// TIA Portal project "机器人" (V14)

(* hardware
DEVICE "S71500/ET200MP station_1"  S7-1500 station
   slot 0: "导轨_0"  Rack  6ES7 590-1***0-0AA0
   slot 1: "PLC_1"  CPU 1516-3 PN/DP  6ES7 516-3AN01-0AB0  V2.1
      slot 3: "CPU 显示_1"  6ES7591-1BA00-0AA0
   slot 2: "DI 32x24VDC HF_1"  DI 32x24VDC HF  6ES7 521-1BL00-0AB0  V2.1
   slot 3: "DQ 32x24VDC/0.5A HF_1"  DQ 32x24VDC/0.5A HF  6ES7 522-1BL01-0AB0  V1.0
   slot 4: "AI 8xU/I/RTD/TC ST_1"  AI 8xU/I/RTD/TC ST  6ES7 531-7KF00-0AB0  V2.1
   slot 5: "AQ 4xU/I ST_1"  AQ 4xU/I ST  6ES7 532-5HD00-0AB0  V2.1
DEVICE "HMI_1"  KTP1200 Basic PN
   slot 0: "KTP1200 Basic PN"  KTP1200 Basic PN  6AV2 123-2MB03-0AX0  14.0.1.0
   slot 1: "HMI_RT_1"  KTP1200 Basic PN  6AV2 123-2MB03-0AX0  14.0.1.0
   slot 5: "HMI_1.IE_CP_1"  PROFINET Interface  14.0.1.0
      slot 1: "PROFINET Interface_1"  PROFINET Interface
         slot 1: "Port_1"  Port
*)

// ===== PLC "PLC_1"  CPU 1516-3 PN/DP =====

VAR_GLOBAL   // PLC tag table "变量表_1"
   "无刷电机传送带传感器1" AT %I0.0 : Bool;   // 检测到有料时值为1
   "无刷电机传送带传感器2" AT %I0.1 : Bool;   // 检测到有料时值为1
   "无刷电机传送带传感器3" AT %I0.2 : Bool;   // 检测到有料时值为1
   "V90传送带传感器1" AT %I0.3 : Bool;   // 检测到有料时值为1
   "V90传送带传感器2" AT %I0.4 : Bool;   // 检测到有料时值为1
   "V90传送带传感器3" AT %I0.5 : Bool;   // 检测到有料时值为1
   "G120传送带物料井检料光纤传感器" AT %I0.6 : Bool;   // 检测到有料时值为1
   "G120传送带物料井推料气缸原位信号" AT %I0.7 : Bool;   // 气缸在原位时值为1
   "G120传送带物料井推料气缸工作位信号" AT %I1.0 : Bool;   // 气缸在工作位时值为1
   "G120传送带末端检料传感器信号" AT %I1.1 : Bool;   // 检测到有料时值为1
   "对射传感器检测信号" AT %I1.2 : Bool;   // 对射传感器之间检测有物体时为1
   "电池底盒气缸原位信号" AT %I1.3 : Bool;   // 气缸在原位时值为1
   "电池底盒气缸工作位信号" AT %I1.4 : Bool;   // 气缸在工作位时值为1
   "输出测试反馈信号" AT %I1.5 : Bool;   // 电池盒装配测试反馈信号
   "前门传感器信号" AT %I1.6 : Bool;   // 前门关闭时值为1
   "后门传感器信号" AT %I1.7 : Bool;   // 后门关闭时值为1
   "机器人输出信号对接1" AT %I2.0 : Bool;   // 可自定义功能例如：急停
   "机器人输出信号对接2" AT %I2.1 : Bool;   // 可自定义功能例如：原位
   "机器人输出信号对接3" AT %I2.2 : Bool;   // 可自定义功能例如：自动
   "机器人输出信号对接4" AT %I2.3 : Bool;   // 可自定义功能例如：就绪
   "机器人输出信号对接5" AT %I2.4 : Bool;   // 可自定义功能例如：完成
   "机器人输出信号对接6" AT %I2.5 : Bool;   // 可自定义功能：待定
   "机器人输出信号对接7" AT %I2.6 : Bool;   // 可自定义功能：待定
   "机器人输出信号对接8" AT %I2.7 : Bool;   // 可自定义功能：待定
   "机器人输出信号对接9" AT %I3.0 : Bool;   // 可自定义功能：待定
   "机器人输出信号对接10" AT %I3.1 : Bool;   // 可自定义功能：待定
   "机器人输出信号对接11" AT %I3.2 : Bool;   // 可自定义功能：待定
   "机器人输出信号对接12" AT %I3.3 : Bool;   // 可自定义功能：待定
   "机器人输出信号对接13" AT %I3.4 : Bool;   // 可自定义功能：待定
   "DI_备用1" AT %I3.5 : Bool;   // DI_备用1
   "DI_备用2" AT %I3.6 : Bool;   // DI_备用2
   "DI_备用3" AT %I3.7 : Bool;   // DI_备用3
END_VAR

VAR_GLOBAL   // PLC tag table "变量表_2"
   "连接传送带电机输出（工作站之间的传送带驱动电机）" AT %Q0.0 : Bool;   // 工作站之间连接传送带电机输出
   "G120传送带物料井推料气缸输出" AT %Q0.1 : Bool;   // 值为1时使气缸推出
   "电池底盒原位气缸输出" AT %Q0.2 : Bool;   // 值为1时使气缸退回
   "电池底盒工作位气缸输出" AT %Q0.3 : Bool;   // 值为1时使气缸推出
   "测试灯输出" AT %Q0.4 : Bool;   // 电池底盒测试灯输出
   "三色灯（绿灯）" AT %Q0.5 : Bool;   // 绿色柱灯
   "三色灯（黄灯）" AT %Q0.6 : Bool;   // 黄色柱灯
   "三色灯（红灯）" AT %Q0.7 : Bool;   // 红色柱灯
   "蜂鸣器" AT %Q1.0 : Bool;   // 值为1时蜂鸣器响
   "无刷电机正转" AT %Q1.1 : Bool;   // 值为1时无刷电机正转
   "无刷电机反转" AT %Q1.2 : Bool;   // 值为1时无刷电机反转
   "无刷电机速度M0" AT %Q1.3 : Bool;   // 无刷电机速度M0
   "无刷电机速度M1" AT %Q1.4 : Bool;   // 无刷电机速度M1
   "备用中继输出1" AT %Q1.5 : Bool;   // 备用中继输出1
   "备用中继输出2" AT %Q1.6 : Bool;   // 备用中继输出2
   "备用中继输出3" AT %Q1.7 : Bool;   // 备用中继输出3
   "机器人输入信号对接1" AT %Q2.0 : Bool;   // 可自定义功能例如：急停
   "机器人输入信号对接2" AT %Q2.1 : Bool;   // 可自定义功能例如：保护回路
   "机器人输入信号对接3" AT %Q2.2 : Bool;   // 可自定义功能例如：程序启动
   "机器人输入信号对接4" AT %Q2.3 : Bool;   // 可自定义功能例如：程序执行
   "机器人输入信号对接5" AT %Q2.4 : Bool;   // 可自定义功能：待定
   "机器人输入信号对接6" AT %Q2.5 : Bool;   // 可自定义功能：待定
   "机器人输入信号对接7" AT %Q2.6 : Bool;   // 可自定义功能：待定
   "机器人输入信号对接8" AT %Q2.7 : Bool;   // 可自定义功能：待定
   "机器人输入信号对接9" AT %Q3.0 : Bool;   // 可自定义功能：待定
   "机器人输入信号对接10" AT %Q3.1 : Bool;   // 可自定义功能：待定
   "机器人输入信号对接11" AT %Q3.2 : Bool;   // 可自定义功能：待定
   "机器人输入信号对接12" AT %Q3.3 : Bool;   // 可自定义功能：待定
   "DO_备用1" AT %Q3.4 : Bool;   // DO_备用1
   "DO_备用2" AT %Q3.5 : Bool;   // DO_备用2
   "DO_备用3" AT %Q3.6 : Bool;   // DO_备用3
   "DO_备用4" AT %Q3.7 : Bool;   // DO_备用4
END_VAR

VAR_GLOBAL   // PLC tag table "变量表_3"
   "M_Safeguards" AT %M10.0 : Bool;   // 安全保护
   "M_E_Stop" AT %M10.1 : Bool;   // 紧急停止
   "M_Start" AT %M10.2 : Bool;   // 启动
   "M_Stop" AT %M10.3 : Bool;   // 停止
   "M_Safe_Confirm" AT %M10.4 : Bool;   // 安全确认
   "M_Ack_E_Stop" AT %M10.5 : Bool;   // 复位紧急停止
   "M_Enable" AT %M10.6 : Bool;   // 使能
   "M_Starting" AT %M10.7 : Bool;   // 启动中
   "M_Edge" AT %M11.0 : Bool;   // 信号沿
   "M_P1" AT %M11.1 : Bool;   // 上升沿寄存器1
END_VAR

FUNCTION "Function" : Void   // FC1, LAD
{ S7_Optimized_Access := 'TRUE' }
VERSION : 0.1
   VAR_TEMP   // added for the SCL form of the ladder/FBD networks
      _w1 : Bool;
   END_VAR
BEGIN

REGION Network 1: 安全保护
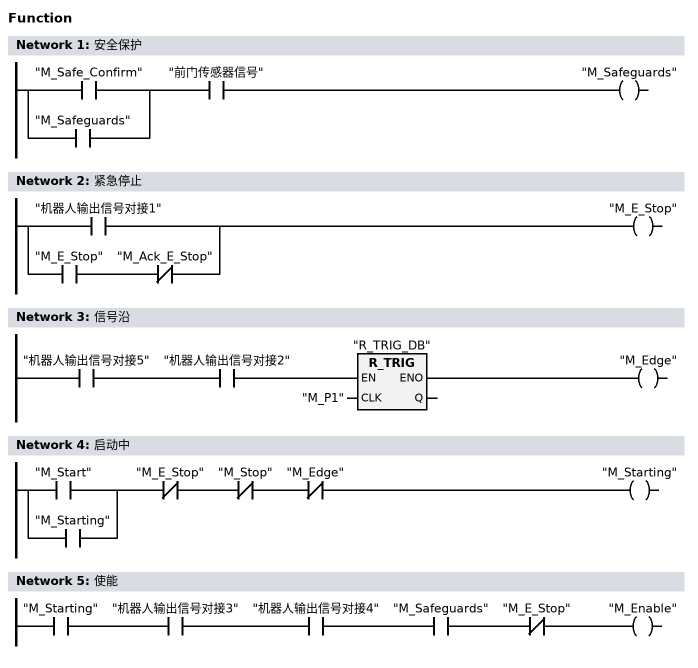
   RUNG wire#powerrail
      Contact( "M_Safe_Confirm" )
      wire#w1
      Contact( "前门传感器信号" )
      Coil( "M_Safeguards" )
   END_RUNG
   RUNG wire#powerrail
      Contact( "M_Safeguards" )
   END_RUNG wire#w1
   // the same network as SCL:
   "M_Safeguards" := ("M_Safe_Confirm" OR "M_Safeguards") AND "前门传感器信号";
END_REGION

REGION Network 2: 紧急停止
   RUNG wire#powerrail
      Contact( "机器人输出信号对接1" )
      wire#w1
      Coil( "M_E_Stop" )
   END_RUNG
   RUNG wire#powerrail
      Contact( "M_E_Stop" )
      I_Contact( "M_Ack_E_Stop" )
   END_RUNG wire#w1
   // the same network as SCL:
   "M_E_Stop" := "机器人输出信号对接1" OR ("M_E_Stop" AND NOT "M_Ack_E_Stop");
END_REGION

REGION Network 3: 信号沿
   // ENO of a box is taken as its EN; it also drops when the box reports an error
   #_w1 := "机器人输出信号对接5" AND "机器人输出信号对接2";
   IF #_w1 THEN
       "R_TRIG_DB"(CLK := "M_P1");   // R_TRIG
   END_IF;
   "M_Edge" := #_w1;
END_REGION

REGION Network 4: 启动中
   RUNG wire#powerrail
      Contact( "M_Start" )
      wire#w1
      I_Contact( "M_E_Stop" )
      I_Contact( "M_Stop" )
      I_Contact( "M_Edge" )
      Coil( "M_Starting" )
   END_RUNG
   RUNG wire#powerrail
      Contact( "M_Starting" )
   END_RUNG wire#w1
   // the same network as SCL:
   "M_Starting" := ("M_Start" OR "M_Starting") AND NOT "M_E_Stop" AND NOT "M_Stop" AND NOT "M_Edge";
END_REGION

REGION Network 5: 使能
   RUNG wire#powerrail
      Contact( "M_Starting" )
      Contact( "机器人输出信号对接3" )
      Contact( "机器人输出信号对接4" )
      Contact( "M_Safeguards" )
      I_Contact( "M_E_Stop" )
      Coil( "M_Enable" )
   END_RUNG
   // the same network as SCL:
   "M_Enable" := "M_Starting" AND "机器人输出信号对接3" AND "机器人输出信号对接4" AND "M_Safeguards" AND NOT "M_E_Stop";
END_REGION
END_FUNCTION

FUNCTION "Light" : Void   // FC2, LAD
{ S7_Optimized_Access := 'TRUE' }
VERSION : 0.1
BEGIN

REGION Network 1: 检测到有料时值为1
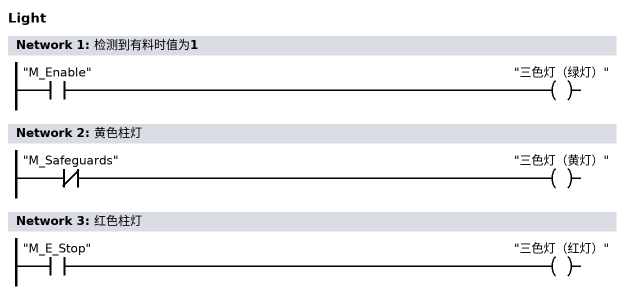
   RUNG wire#powerrail
      Contact( "M_Enable" )
      Coil( "三色灯（绿灯）" )
   END_RUNG
   // the same network as SCL:
   "三色灯（绿灯）" := "M_Enable";
END_REGION

REGION Network 2: 黄色柱灯
   RUNG wire#powerrail
      I_Contact( "M_Safeguards" )
      Coil( "三色灯（黄灯）" )
   END_RUNG
   // the same network as SCL:
   "三色灯（黄灯）" := NOT "M_Safeguards";
END_REGION

REGION Network 3: 红色柱灯
   RUNG wire#powerrail
      Contact( "M_E_Stop" )
      Coil( "三色灯（红灯）" )
   END_RUNG
   // the same network as SCL:
   "三色灯（红灯）" := "M_E_Stop";
END_REGION
END_FUNCTION

FUNCTION "Robot" : Void   // FC3, LAD
{ S7_Optimized_Access := 'TRUE' }
VERSION : 0.1
BEGIN

REGION Network 1: 可自定义功能例如：急停
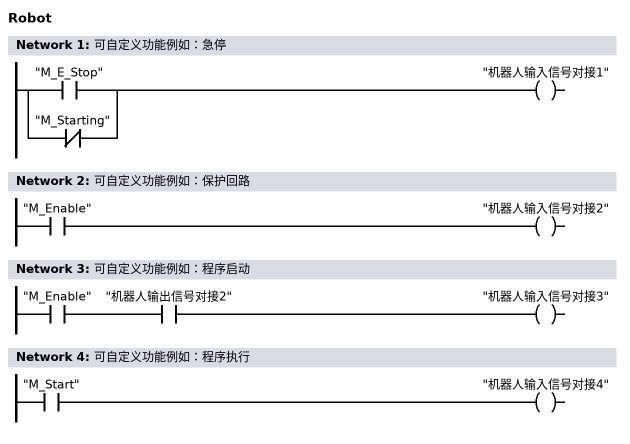
   RUNG wire#powerrail
      Contact( "M_E_Stop" )
      wire#w1
      Coil( "机器人输入信号对接1" )
   END_RUNG
   RUNG wire#powerrail
      I_Contact( "M_Starting" )
   END_RUNG wire#w1
   // the same network as SCL:
   "机器人输入信号对接1" := "M_E_Stop" OR NOT "M_Starting";
END_REGION

REGION Network 2: 可自定义功能例如：保护回路
   RUNG wire#powerrail
      Contact( "M_Enable" )
      Coil( "机器人输入信号对接2" )
   END_RUNG
   // the same network as SCL:
   "机器人输入信号对接2" := "M_Enable";
END_REGION

REGION Network 3: 可自定义功能例如：程序启动
   RUNG wire#powerrail
      Contact( "M_Enable" )
      Contact( "机器人输出信号对接2" )
      Coil( "机器人输入信号对接3" )
   END_RUNG
   // the same network as SCL:
   "机器人输入信号对接3" := "M_Enable" AND "机器人输出信号对接2";
END_REGION

REGION Network 4: 可自定义功能例如：程序执行
   RUNG wire#powerrail
      Contact( "M_Start" )
      Coil( "机器人输入信号对接4" )
   END_RUNG
   // the same network as SCL:
   "机器人输入信号对接4" := "M_Start";
END_REGION
END_FUNCTION

ORGANIZATION_BLOCK "Main"   // OB1, LAD, ProgramCycle
TITLE = "Main Program Sweep (Cycle)"
{ S7_Optimized_Access := 'TRUE' }
VERSION : 0.1
   VAR_INPUT
      Initial_Call : Bool;   // Initial call of this OB
      Remanence : Bool;   // =True, if remanent data are available
   END_VAR
BEGIN

REGION Network 1
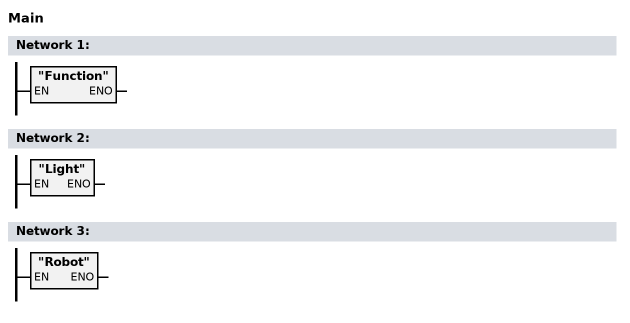
   RUNG wire#powerrail
      "Function"()
   END_RUNG
   // the same network as SCL:
   "Function"();
END_REGION

REGION Network 2
   RUNG wire#powerrail
      "Light"()
   END_RUNG
   // the same network as SCL:
   "Light"();
END_REGION

REGION Network 3
   RUNG wire#powerrail
      "Robot"()
   END_RUNG
   // the same network as SCL:
   "Robot"();
END_REGION
END_ORGANIZATION_BLOCK

(* ===== HMI "HMI_RT_1" =====
system functions are stored by id; their names below are inferred from use
connection "HMI_连接_1": ETHERNET, SMART_S7_1500_OMS

HMI tags "默认变量表"
   "Tag_ScreenNumber" : UInt, internal
   "机器人输出信号对接1" : Bool = PLC 机器人输出信号对接1 AT %I2.0, 1 s
   "机器人输出信号对接2" : Bool = PLC 机器人输出信号对接2 AT %I2.1, 1 s
   "机器人输出信号对接3" : Bool = PLC 机器人输出信号对接3 AT %I2.2, 1 s
   "机器人输出信号对接4" : Bool = PLC 机器人输出信号对接4 AT %I2.3, 1 s
   "M_Starting" : Bool = PLC M_Starting AT %M10.7, 1 s
   "M_Start" : Bool = PLC M_Start AT %M10.2, 1 s
   "M_Stop" : Bool = PLC M_Stop AT %M10.3, 1 s
   "M_Safeguards" : Bool = PLC M_Safeguards AT %M10.0, 1 s
   "M_Safe_Confirm" : Bool = PLC M_Safe_Confirm AT %M10.4, 1 s
   "M_E_Stop" : Bool = PLC M_E_Stop AT %M10.1, 1 s
   "M_Ack_E_Stop" : Bool = PLC M_Ack_E_Stop AT %M10.5, 1 s
   "M_Enable" : Bool = PLC M_Enable AT %M10.6, 1 s

screen "根画面" 1280x800, template "Template_1"
   on GenerateScreen: SetTag("Tag_ScreenNumber", 1)
   TextField "HmiScreenItemData" at 128,384 size 1024x27; Text '欢迎进入 HMI_1 (KTP1200 Basic+ PN)！'
   GraphicView "图形视图_1" at 1,155 size 1279x645; Picture "station"
   TextField "文本域_1" at 1072,12 size 101x27; Text '控制面板'
   Circle "圆_1" at 1055,70 size 49x49
      Appearance <- "机器人输出信号对接1"
   TextField "文本域_2" at 1038,140 size 95x21; Text '机器人急停'
   Circle "圆_2" at 1172,68 size 49x49
      Appearance <- "机器人输出信号对接2"
   Circle "圆_3" at 1057,185 size 49x49
      Appearance <- "机器人输出信号对接3"
   Circle "圆_4" at 1174,182 size 49x49
      Appearance <- "机器人输出信号对接4"
   TextField "文本域_3" at 1151,140 size 95x21; Text '机器人复位'
   TextField "文本域_4" at 1038,250 size 95x21; Text '机器人自动'
   TextField "文本域_5" at 1151,250 size 95x21; Text '机器人就绪'
   Button "按钮_1" at 1037,290 size 87x39; TextOff '启动'
      Appearance <- "M_Starting"
      on Press: SetBit("M_Start")
      on Release: ResetBit("M_Start")
   Button "按钮_2" at 1151,290 size 87x39; TextOff '停止'
      on Press: SetBit("M_Stop")
      on Release: ResetBit("M_Stop")
   Button "按钮_3" at 1038,345 size 87x39; TextOff '确认安全'
      Appearance <- "M_Safeguards"
      on Press: SetBit("M_Safe_Confirm")
      on Release: ResetBit("M_Safe_Confirm")
   Button "按钮_4" at 1151,345 size 87x39; TextOff '复位急停'
      Appearance <- "M_E_Stop"
      on Press: SetBit("M_Ack_E_Stop")
      on Release: ResetBit("M_Ack_E_Stop")
   Button "按钮_5" at 1091,403 size 100x43; TextOff '使能中'
      Appearance <- "M_Enable"
      Visibility <- "M_Enable"

Template "Template_1" 1280x800
   Button "退出" at 1182,752 size 67x47; TextOff '退出'; PictureOff "ExitRuntime_KTP1200_Basic_PN_TR"; PictureOn "ExitRuntime_KTP1200_Basic_PN_TR"
      on Release: StopRuntime(0)
   Button "Template_Button" at 1054,752 size 67x47; TextOff 'Text'
   Button "Template_Button_1" at 926,752 size 67x47; TextOff 'Text'
   Button "Template_Button_2" at 798,752 size 67x47; TextOff 'Text'
   Button "Template_Button_3" at 670,752 size 67x47; TextOff 'Text'
   Button "Template_Button_4" at 542,752 size 67x47; TextOff 'Text'
   Button "Template_Button_5" at 414,752 size 67x47; TextOff 'Text'
   Button "Template_Button_6" at 286,752 size 67x47; TextOff 'Text'
   Button "报警" at 158,752 size 67x47; TextOff '报警'; PictureOff "AlarmDisplay_KTP1200_Basic_PN_TR"; PictureOn "AlarmDisplay_KTP1200_Basic_PN_TR"
      on Release: function_ef3f5d25("报警窗口_Unacknowledged", -1)
   Button "起始画面" at 30,752 size 67x47; TextOff '起始画面'; PictureOff "NavigateHome_KTP1200_Basic_PN_TR"; PictureOn "NavigateHome_KTP1200_Basic_PN_TR"
      on Release: ActivateScreen("根画面", 0)
   SymbolicIOField "Symbolic_IO_Field_Screen" at 87,9 size 1086x30; TextOff '0'; TextOn '1'; TextList "TextList_ScreenNames"
      ProcessValue <- "Tag_ScreenNumber"
      on Change: ActivateScreenByNumber("Tag_ScreenNumber", 0)
   DateTimeField "HmiScreenItemData" at 1175,24 size 105x24
   DateTimeField "HmiScreenItemData_1" at 1175,0 size 105x24
   GraphicView "Logo" at 0,0 size 85x48; Picture "HMI_1 的 Logo"
*)